// ---- POUs/Prototypes/TcoSequencer/TcoSequencerBase.TcPOU
(*~
        <docu>
            <summary>
                Provides basic sequential control, including step mode, which allows to run the sequence step-by-step, steping forward and steping backward.
            </summary>
        </docu>
~*)
FUNCTION_BLOCK ABSTRACT TcoSequencerBase EXTENDS TcoStateExtendible IMPLEMENTS ITcoSequencer, ITcoCoordinator
VAR CONSTANT
    MinStepID : INT := -32767;
    MaxStepID : INT := 32766;
    RESTORE_STEP_ID : INT := 32766;
END_VAR
VAR
    (*~
    <docu>
        <summary>
            Holds the status information about current step.
        </summary>
        <remarks>
            <para>
                See <see cref="StepDetails"/> for detailed description.
            </para>
        </remarks>
    </docu>
~*)
    {attribute addProperty Name "<#Current step#>"}
    _currentStep : StepDetails;
    (*~
    <docu>
        <summary>
            True if an error occurs in the sequence. Detailed cause of this error is described by the _sequencerErrorId.
        </summary>
        <remarks>
            <para>
                See <see cref="PlcDocu.TcoCore.TcoSequencer._sequencerErrorId"/> for detailed description.
            </para>
        </remarks>
    </docu>
~*)
    {attribute addProperty Name "<#Sequencer error#>"}
    {attribute clr [ReadOnly()]}
    _sequencerHasError : BOOL;
    (*~
    <docu>
        <summary>
            Describes cause of the sequencer error.
        </summary>
        <remarks>
            <para>
                See <see cref="TcoCore.eSequencerError"/> for detailed description.
            </para>
        </remarks>
    </docu>
~*)
    {attribute addProperty Name "<#Sequencer error ID#>"}
    {attribute clr [ReadOnly()]}
    _sequencerErrorId : eSequencerError := eSequencerError.noError;
    (*~
    <docu>
        <summary>
            Handles changing the sequencer mode (Cyclic, Step).
        </summary>
    </docu>
~*)
    _modeController : TcoSequencerModeController(THIS^);
    (*~
    <docu>
        <summary>
            Elapsed time of presently running sequence cycle.
        </summary>
    </docu>
~*)
    {attribute addProperty Name "<#Sequence cycle elapsed time#>"}
    _SequenceElapsedTime : TIME;
    (*~
    <docu>
        <summary>
            Elapsed time of the currently executing step.
        </summary>
    </docu>
~*)
    {attribute addProperty Name "<Current step time#>"}
    _StepElapsedTime : TIME;
    (*~
    <docu>
        <summary>
            Total time of the last sequence cycle.
        </summary>
    </docu>
~*)
    {attribute addProperty Name "<#Total sequence time#>"}
    _LastCycleTime : TIME;
END_VAR
VAR
    {attribute 'hide'}
    _isFirstStepEntry : BOOL;
    {attribute 'hide'}
    _theOrderOfTheCurrentlyEvaluatedStep : UINT;
    {attribute 'hide'}
    _theOrderOfTheCurrentlyExecutedStep : UINT;
    {attribute 'hide'}
    _theOrderOfThePreviouslyExecutedStep : UINT;
    {attribute 'hide'}
    _IdOfThePreviouslyExecutedStep : INT;
    {attribute 'hide'}
    _numberOfStepsInSequence : UINT;
    {attribute 'hide'}
    _previousNumberOfStepsInSequence : UINT;
    {attribute 'hide'}
    _stepCounter : UINT;
    {attribute 'hide'}
    _requestStepActive : BOOL;
    {attribute 'hide'}
    _requestedStepId : INT := MinStepID - 1;
    {attribute 'hide'}
    _cycleTimer : TON;
    {attribute 'hide'}
    _StepTimer : TON;
    {attribute 'hide'}
    _requestStepCycle : UINT;
    {attribute 'hide'}
    _StepIdChanged : BOOL;
    {attribute 'hide'}
    _StepOrderChanged : BOOL;
    {attribute 'hide'}
    _ChangeStepIdFrom : INT;
    {attribute 'hide'}
    _ChangeStepIdTo : INT;
    {attribute 'hide'}
    _ChangeStepOrderFrom : UINT;
    {attribute 'hide'}
    _ChangeStepOrderTo : UINT;
    {attribute 'hide'}
    _stepIdUniquenessChecked : BOOL := FALSE;
    {attribute 'hide'}
    _StepIdUniquenessControlState : eStepIdUniquenessControlState;
    {attribute 'hide'}
    _StepIdUniquenessStartCycleCount : ULINT;
    {attribute 'hide'}
    _checkStepIdRequestedInStepMode : BOOL;
    {attribute 'hide'}
    _restoringSequence : BOOL;
    {attribute 'hide'}
    _controlledStepIndex : UINT;
END_VAR
VAR
    {attribute 'hide'}
    _pPreviusSteps : POINTER TO INT;
END_VAR
VAR
    {attribute 'hide'}
    _lastOpeningCycle : ULINT;
    {attribute 'hide'}
    _lastClosingCycle : ULINT;
END_VAR
VAR
    _observer : ITcoSequencerObserver;
    {attribute 'hide'}
    _observerDummy : TcoTcoSequencerObserverDummy(THIS^);
END_VAR

METHOD PUBLIC FINAL ActivateDeveloperChecks
VAR_INPUT
END_VAR
IF (_StepIdUniquenessControlState = eStepIdUniquenessControlState.Deactivated) THEN
    _StepIdUniquenessControlState := eStepIdUniquenessControlState.Requested;
END_IF
END_METHOD

(*~
    <docu>
        <summary>
            Performs the check of the ```StepId``` of the currently executed step.
            <remarks>
                <note type="important">
                    The StepId of each step in the sequence must be unique throughout the complete sequence, and it must not be changed.
                    ```StepId``` sould be assigned as a number literal or a constant.
                </note>
            </remarks>
        </summary>
    </docu>
~*)
METHOD PRIVATE CheckStepId : BOOL
VAR_INPUT
    inStepID : INT;
    inStepModeActive : BOOL;
    inStepInRunning : BOOL;
END_VAR
CheckStepID := TRUE;

IF (_StepIdUniquenessControlState = eStepIdUniquenessControlState.Done) THEN
    IF ((_IdOfThePreviouslyExecutedStep <> inStepID) AND NOT _isFirstStepEntry AND (NOT inStepModeActive OR inStepInRunning)) THEN
        IF (_theOrderOfTheCurrentlyExecutedStep = 0) AND (_theOrderOfTheCurrentlyEvaluatedStep = 0) AND (_IdOfThePreviouslyExecutedStep = 0) THEN
            _IdOfThePreviouslyExecutedStep := inStepID;
        ELSIF NOT _StepIdChanged AND NOT _StepOrderChanged THEN
            _StepIdChanged := TRUE;
            _ChangeStepIdFrom := _IdOfThePreviouslyExecutedStep;
            _ChangeStepIdTo := inStepID;
            CheckStepID := FALSE;
        END_IF;
    END_IF
END_IF
END_METHOD

(*~
    <docu>
        <summary>
            Gets the information about the current step.
        </summary>
    </docu>
~*)
PROPERTY CurrentStep : REFERENCE TO StepDetails
GET
CurrentStep REF= _currentStep;
END_GET
END_PROPERTY

METHOD PUBLIC FINAL DeactivateDeveloperChecks
VAR_INPUT
END_VAR
_StepIdUniquenessControlState := eStepIdUniquenessControlState.Deactivated;
END_METHOD

{attribute 'hide'}
METHOD FB_init : BOOL
VAR_INPUT
    bInitRetains : BOOL; // if TRUE, the retain variables are initialized (warm start / cold start)
    bInCopyCode : BOOL; // if TRUE, the instance afterwards gets moved into the copy code (online change)
    ParentObject : ITcoObject;
    AutoRestoreMode : eRestoreMode;
END_VAR
END_METHOD

(*~
    <docu>
        <summary>
            Implicit call of this method is ensured by calling the method Run().
            It must not be called explicitely by consumer code in derived blocks.
            <remarks>
                <note type="important">
                    Do not call this method explicitly.
                </note>
            </remarks>
        </summary>
    </docu>
~*)
METHOD INTERNAL FINAL i_Close
_lastClosingCycle := Context.StartCycleCount;

IF _sequencerHasError THEN
    OnSequencerError(_sequencerErrorId);
END_IF

_previousNumberOfStepsInSequence := _numberOfStepsInSequence;
Context.Environment.Messaging.Suspend();

IF _modeController._stepIn.Done THEN
    _modeController._stepIn.Restore();
END_IF

Context.Environment.Messaging.Resume();
_restoringSequence := FALSE;
END_METHOD

(*~
    <docu>
        <summary>
            <para>
                Completes the sequencer, and return the sequencer pointer to the first step in the seuqence.
                Method is typically called inside the last step of the sequence.
            </para>
        </summary>
    </docu>
~*)
METHOD PROTECTED FINAL i_CompleteSequence
_theOrderOfTheCurrentlyExecutedStep := 0;
_LastCycleTime := _SequenceElapsedTime;
_cycleTimer(IN := FALSE, PT := T#0S);
_currentStep.Status := eStepStatus.Done;
OnSequenceCompleted();
OnStepCompleted();
Context.Environment.Messaging.Suspend();
_modeController._stepForward.Restore();
_modeController._stepBackward.Restore();
_modeController._stepIn.Restore();
Context.Environment.Messaging.Resume();
END_METHOD

(*~
    <docu>
        <summary>
            Completes the execution of the current step and moves the sequencer pointer to the next step in order of execution.
            The call returns `ITcoObjectRestorer` that allows to restore object upon step completition.
        </summary>
        <returns></returns>
    </docu>
~*)
METHOD PROTECTED FINAL i_CompleteStep : ITcoObjectRestorer
Messenger.Build()
    .Append('Leaving step id: ')
    .AppendAny(_currentStep.ID)
    .Append(' [')
    .Append(_currentStep.Description)
    .Append('] : ')
    .AppendAny(_theOrderOfTheCurrentlyExecutedStep)
    .As().AsTrace();

_theOrderOfTheCurrentlyExecutedStep := _theOrderOfTheCurrentlyExecutedStep + 1;
_currentStep.Status := eStepStatus.Done;
OnStepCompleted();
_modeController._stepIn.DoneWhen(_modeController._stepIn.Execute());
i_CompleteStep := THIS^;
END_METHOD

(*~
    <docu>
        <summary>
            Implicit calling of this method is ensured by calling the method Run().
            It must not be called explicitely by consumer code in derived blocks.
            <remarks>
                <note type="important">
                    Do not call this method explicitly.
                </note>
            </remarks>
        </summary>
    </docu>
~*)
METHOD INTERNAL FINAL i_Open
VAR
    _message : STRING(254);
END_VAR
_theOrderOfTheCurrentlyEvaluatedStep := 0;

IF _requestStepActive AND
    _requestedStepId <> (MinStepID - 1) AND
    (_modeController.Mode <> eSequencerMode.StepMode OR _modeController._stepIn.Busy OR _checkStepIdRequestedInStepMode) THEN
    _requestStepCycle := _requestStepCycle + 1;
ELSE
    _requestStepCycle := 0;
END_IF

IF _requestStepCycle > 1 AND NOT _sequencerHasError THEN
    _sequencerErrorId := eSequencerError.StepWithRequestedIdDoesNotExists;
    _message := CONCAT('REQUESTED STEP_ID: ', INT_TO_STRING(_requestedStepId));
    _message := CONCAT(_message, ' DOES NOT EXIST');
    _currentStep.Description := _message;
    _currentStep.Status := eStepStatus.Error;
    THIS^.Messenger.Post(_message, eMessageCategory.ProgrammingError);
    _sequencerHasError := TRUE;
END_IF

IF _StepIdUniquenessControlState = eStepIdUniquenessControlState.NotYetStarted OR
    _StepIdUniquenessControlState = eStepIdUniquenessControlState.Requested THEN
    _StepIdUniquenessControlState := eStepIdUniquenessControlState.Started;
END_IF;

_restoringSequence := FALSE;
_lastOpeningCycle := Context.StartCycleCount;
END_METHOD

(*~
    <docu>
        <summary>
            Terminates the currently executed step and set the sequencer's pointer to the step with Id that corresponds to ```inRequestedStepID``` parameter.
            When the order of the requested step is higher than the order of the currently finished step (the requested step is "after" the current one)
            the requested step is started in the same context cycle.
            When the order of the requested step is lower than the order of the currently finished step (the requested step is "before" the current one)
            the requested step is started in the next context cycle.
            If the requested step is not found even in the next context cycle, the sequencer enters error state ```StepWithRequestedIdDoesNotExists```.
            <para>
                See <see cref="TcoCore.eSequencerError"/> for detailed description.
            </para>
        </summary>
    </docu>
~*)
METHOD PROTECTED FINAL i_RequestStep : ITcoSequencer
VAR_INPUT
    (*~
        <docu>
            <summary>
                StepId of the step to be executed.
            </summary>
        </docu>
    ~*)
    inRequestedStepID : INT := MinStepID - 1;
END_VAR
VAR
    _message : STRING(254);
END_VAR
_modeController._stepIn.Restore();
_currentStep.Status := eStepStatus.Done;
_checkStepIdRequestedInStepMode := TRUE;

IF (inRequestedStepID <> (MinStepID - 1)) THEN
    IF _requestedStepId <> (MinStepID - 1) THEN
        IF NOT _sequencerHasError THEN
            _sequencerErrorId := eSequencerError.MultipleRequestStepMethodCall;
            _message := CONCAT('REQUESTED STEP_ID: ', INT_TO_STRING(inRequestedStepID));
            _message := CONCAT(_message, ' HAS BEEN REQUIRED, WHILE PREVIOUS REQUESTED STEP_ID: ');
            _message := CONCAT(_message, INT_TO_STRING(_requestedStepId));
            _message := CONCAT(_message, ' HAS NOT BEEN YET PERFORMED!');
            _currentStep.Description := _message;
            _currentStep.Status := eStepStatus.Error;
            THIS^.Messenger.Post(_message, eMessageCategory.ProgrammingError);
            _sequencerHasError := TRUE;
        END_IF
    ELSE
        _requestStepCycle := 0;
        _requestedStepId := inRequestedStepID;
        _requestStepActive := TRUE;
    END_IF
END_IF;

Messenger.Build()
    .Append('Leaving step id: ')
    .AppendAny(_currentStep.ID)
    .Append(' [')
    .Append(_currentStep.Description)
    .Append('] : ')
    .AppendAny(_theOrderOfTheCurrentlyExecutedStep)
    .As().AsTrace();

Messenger.Build().Append('Reqesting step id jump to: ').AppendAny(inRequestedStepID).As().AsTrace();
i_RequestStep := THIS^;
END_METHOD

(*~
    <docu>
        <summary>
                Step of the sequence.
                <note type="important">
                    Make sure you do not use the value of `32766` for the step id. This value is reserved for the restore step.
                <note>
        </summary>
        <returns>
            True when step with given `StepId` is in order of the execution; the step is enabled and the sequencer is in the cyclic mode.
            True when step with given `StepId` is in order of the execution; the step is enabled, the sequencer is in the step mode and StepIn() method has been triggered.
        </returns>
    </docu>
~*)
METHOD PROTECTED FINAL i_Step : BOOL
VAR_INPUT
    (*~
    <docu>
        <summary>
            StepId of the current step.
            <remarks>
                <note type="important">
                    This number must be unique throughout the complete sequence.
                    It must be a constant or numerical literal and it must not change during the life-time of the sequencer.
                </note>
                <note type="important">
                    Make sure you do not use the value of `32766` for the step id. This value is reserved for the restore step.
                <note>
            </remarks>
        </summary>
    </docu>
~*)
    inStepID : INT;
    (*~
    <docu>
        <summary>
            If this value is false, step body is not executed and execution is moved to the next enabled step.
        </summary>
    </docu>
~*)
    inEnabled : BOOL;
    (*~
    <docu>
        <summary>
            Step description text.
        </summary>
    </docu>
~*)
    inStepDescription : STRING(254);
END_VAR
VAR
    _message : STRING(254);
    _isInOrderOfExecution : BOOL;
    _stepModeActive : BOOL;
    _stepInExecuting : BOOL;
END_VAR
i_Step := FALSE;

IF inStepID < MinStepID THEN
    _message := CONCAT('STEP_ID TOO LOW: ', INT_TO_STRING(inStepID));
    _message := CONCAT(_message, '! MINIMAL VALUE POSSIBLE: ');
    _message := CONCAT(_message, INT_TO_STRING(MinStepID));
    _message := CONCAT(_message, '!!!');
    _currentStep.Description := _message;
    _currentStep.Status := eStepStatus.Error;
    THIS^.Messenger.Post(_message, eMessageCategory.ProgrammingError);
    _sequencerErrorId := eSequencerError.StepIdTooLow;
    _sequencerHasError := TRUE;
ELSIF inStepID > MaxStepID THEN
    _message := CONCAT('STEP_ID TOO HIGH: ', INT_TO_STRING(inStepID));
    _message := CONCAT(_message, '! MAXIMAL VALUE POSSIBLE: ');
    _message := CONCAT(_message, INT_TO_STRING(MaxStepID));
    _message := CONCAT(_message, '!!!');
    _currentStep.Description := _message;
    _currentStep.Status := eStepStatus.Error;
    THIS^.Messenger.Post(_message, eMessageCategory.ProgrammingError);
    _sequencerErrorId := eSequencerError.StepIdTooHigh;
    _sequencerHasError := TRUE;
ELSIF NOT _sequencerHasError THEN
    i_Step := StepInternal(inStepID, inEnabled, inStepDescription);
END_IF;

Observer.Observe(inIsStepActive := i_Step,
    inCurrentStepOrder := _theOrderOfTheCurrentlyExecutedStep,
    inID := inStepID,
    inOrder := _theOrderOfTheCurrentlyEvaluatedStep - 1,
    inEnabled := inEnabled,
    inDescription := inStepDescription,
    inStatus := _currentStep.Status,
    inDuration := _currentStep.Duration,
    inStepCount := _numberOfStepsInSequence);
END_METHOD

(*~
    <docu>
        <summary>
            Completes the actually running step, when the `inCondition` parameter is `TRUE`.
            Method is typically called inside a step as the transition method.
        </summary>
    </docu>
~*)
METHOD PROTECTED FINAL i_StepCompleteWhen
VAR_INPUT
    (*~
    <docu>
        <summary>
            The condition under which the step is completed.
        </summary>
    </docu>
~*)
    inCondition : BOOL;
END_VAR
IF (inCondition) THEN
    THIS^.i_CompleteStep();
END_IF
END_METHOD

(*~
    <docu>
        <summary>
            Gets `true` on the first entry into new state.
        </summary>
    </docu>
~*)
PROPERTY IsFreshState : BOOL
GET
IsFreshState := _isFirstStepEntry;
END_GET
END_PROPERTY

(*~
    <docu>
        <summary>
            Performs the check of the uniqueness of `inStepId` in the sequence.
            <remarks>
                <note type="important">
                    The StepId of each step in the sequence must be unique throughout the complete sequence, and it must not be changed.
                </note>
            </remarks>
        </summary>
    </docu>
~*)
METHOD PRIVATE IsStepIdUnique
VAR_INPUT
    (*~
    <docu>
        <summary>
            StepId to be checked for uniqueness.
        </summary>
    </docu>
~*)
    inStepID : INT;
END_VAR
VAR
    _i : UINT;
    _hiIndex : UINT;
    _pUid : INT;
    _pNewSteps : POINTER TO INT;
    _message : STRING(254);
END_VAR
//Change number of the steps in sequence detected
IF (_numberOfStepsInSequence <> _previousNumberOfStepsInSequence) AND
    _previousNumberOfStepsInSequence > 0 AND
    _stepIdUniquenessChecked AND
    (
    _StepIdUniquenessControlState = eStepIdUniquenessControlState.NotYetStarted OR _StepIdUniquenessControlState = eStepIdUniquenessControlState.Done
    ) THEN
    _StepIdUniquenessControlState := eStepIdUniquenessControlState.Requested;
END_IF

IF (_StepIdUniquenessControlState >= eStepIdUniquenessControlState.Started AND _StepIdUniquenessControlState < eStepIdUniquenessControlState.Done)
    THEN
    //If new PLC cycle was performed, step id uniqueness control is done
    IF _StepIdUniquenessControlState = eStepIdUniquenessControlState.Running AND
        THIS^.Context.StartCycleCount >= _StepIdUniquenessStartCycleCount + 1 THEN
        _stepIdUniquenessChecked := TRUE;
        _StepIdUniquenessControlState := eStepIdUniquenessControlState.Done;
        _numberOfStepsInSequence := _controlledStepIndex + 1;
    END_IF

    //If step id uniqueness control is finished, clear dynamic arrays
    IF _StepIdUniquenessControlState >= eStepIdUniquenessControlState.Done THEN
        IF (_pPreviusSteps <> 0) THEN
            __DELETE(_pPreviusSteps);
        END_IF

        IF (_pNewSteps <> 0) THEN
            __DELETE(_pNewSteps);
        END_IF

        RETURN;
    END_IF

    //First call with the very first step of the sequence
    IF _StepIdUniquenessControlState = eStepIdUniquenessControlState.Started THEN
        _StepIdUniquenessStartCycleCount := THIS^.Context.StartCycleCount;
        _controlledStepIndex := 0;

        //It should not exists, if yes delete and create again
        IF (_pPreviusSteps <> 0) THEN
            __DELETE(_pPreviusSteps);
        END_IF

        _pPreviusSteps := __NEW(UINT, 1);
        //Stores first StepId
        _pPreviusSteps[0] := inStepID;
        _StepIdUniquenessControlState := eStepIdUniquenessControlState.Running;
    ELSIF _StepIdUniquenessControlState = eStepIdUniquenessControlState.Running THEN
        // Increment order of the currently controlled step
        _controlledStepIndex := _controlledStepIndex + 1;

        IF (_pNewSteps <> 0) THEN
            __DELETE(_pNewSteps);
        END_IF

        _pNewSteps := __NEW(UINT, (_controlledStepIndex + 1));
        //Compare with previous Steps and copy previous Steps to new array
        _hiIndex := _controlledStepIndex - 1;

        FOR _i := 0 TO _hiIndex DO
            _pUid := _pPreviusSteps[_i];

            IF inStepID = _pUid THEN
                IF NOT _sequencerHasError THEN
                    _sequencerErrorId := eSequencerError.NotUniqueStepId;
                    _message := CONCAT('ERROR NOT UNIQUE STEP_ID ', INT_TO_STRING(inStepID));
                    _currentStep.Description := _message;
                    _currentStep.Status := eStepStatus.Error;
                    THIS^.Messenger.Post(_message, eMessageCategory.ProgrammingError);
                    _sequencerHasError := TRUE;
                    _StepIdUniquenessControlState := eStepIdUniquenessControlState.Error;
                    RETURN;
                END_IF
            ELSE
                _pNewSteps[_i] := _pPreviusSteps[_i];
            END_IF
        END_FOR
        //Store new StepId
        _pNewSteps[_controlledStepIndex] := inStepID;

        //Delete and create again
        IF (_pPreviusSteps <> 0) THEN
            __DELETE(_pPreviusSteps);
        END_IF

        _pPreviusSteps := __NEW(UINT, (_controlledStepIndex + 1));
        //Copy
        _hiIndex := _controlledStepIndex;

        FOR _i := 0 TO _hiIndex DO
            _pPreviusSteps[_i] := _pNewSteps[_i];
        END_FOR

        IF (_pNewSteps <> 0) THEN
            __DELETE(_pNewSteps);
        END_IF
    END_IF

    _numberOfStepsInSequence := _controlledStepIndex + 1;
END_IF
END_METHOD

(*~
    <docu>
        <summary>
            Main method of the sequener. Custom code needs to be placed here. The sequencer is executed by call of **Instance.Run()** method.
            This method is abstract, and it must be overridden in derived block.
        </summary>
    </docu>
~*)
METHOD PROTECTED ABSTRACT Main : BOOL
END_METHOD

(*~
    <docu>
        <summary>
            Handles changing the sequencer mode (Cyclic, Step).
        </summary>
    </docu>
~*)
PROPERTY ModeController : ITcoSequencerModeController
GET
ModeController := _modeController;
END_GET
END_PROPERTY

{attribute 'hide'}
{attribute 'obsolete' := 'You should access `MoveNext` via `ITcoCoordinator` interface.'}
METHOD PUBLIC MoveNext : BOOL
i_CompleteStep();
END_METHOD

(*~
    <docu>
        <summary>
            Get or sets the observer for this instance of the sequencer.
        </summary>
    </docu>
~*)
PROPERTY Observer : ITcoSequencerObserver
GET
IF (_observer <> 0) THEN
    Observer := _observer;
ELSE
    Observer := _observerDummy;
END_IF
END_GET
SET
_observer := Observer;
END_SET
END_PROPERTY

(*~
    <docu>
        <summary>
            Ensures that after each download, StepId uniqueness check is performed.
            <remarks>
                <note type="important">
                    Do not call this method explicitly.
                </note>
            </remarks>
        </summary>
    </docu>
~*)
{attribute 'call_after_online_change_slot' := '200'}
METHOD PRIVATE OnlineChange
IF _stepIdUniquenessChecked AND (_StepIdUniquenessControlState <> eStepIdUniquenessControlState.Deactivated) THEN
    _StepIdUniquenessControlState := eStepIdUniquenessControlState.Requested;
END_IF;
END_METHOD

(*~
    <docu>
        <summary>
            This method is called on sequence restore.
            This method can be overridden in derived block with a custom logic.
        </summary>
    </docu>
~*)
METHOD PROTECTED OnRestore
END_METHOD

(*~
    <docu>
        <summary>
            This method is called on sequence completion (the sequencer's last step was completed).
            This method can be overridden in derived block with a custom logic.
        </summary>
    </docu>
~*)
METHOD PROTECTED OnSequenceCompleted
END_METHOD

(*~
    <docu>
        <summary>
            This method is called when sequence enters error state. The method is called until the error is cleared.
            This method can be overridden in derived block with a custom logic.
        </summary>
    </docu>
~*)
METHOD PROTECTED OnSequencerError
VAR_INPUT
    inErrorId : eSequencerError;
END_VAR
END_METHOD

METHOD PROTECTED OnStateChange
VAR_INPUT
    PreviousState : INT;
    NewState : INT;
END_VAR
END_METHOD

(*~
    <docu>
        <summary>
            This method is executed upon step completion.
            This method can be overridden in derived block by custom logic.
        </summary>
    </docu>
~*)
METHOD PROTECTED OnStepCompleted
END_METHOD

(*~
    <docu>
        <summary>
            <para>
                This method resets the sequencer.
                Method is typically called before starting the sequence or after error has occured in the sequence.
            </para>
        </summary>
    </docu>
~*)
METHOD PUBLIC Restore : ITcoRestorable
_restoringSequence := TRUE;
_lastClosingCycle := 0;
_lastOpeningCycle := 0;
StepChanged(0);
_requestStepActive := FALSE;
_requestedStepId := MinStepID - 1;
_requestStepCycle := 0;
_sequencerHasError := FALSE;
_sequencerErrorId := eSequencerError.noError;
_currentStep.Description := '--------------------------';
_currentStep.ID := 0;
_currentStep.Order := 0;
_currentStep.Status := eStepStatus.None;
_currentStep.Duration := T#0S;
_stepCounter := 0;
_IdOfThePreviouslyExecutedStep := 0;
_numberOfStepsInSequence := 0;
_previousNumberOfStepsInSequence := 0;
_theOrderOfTheCurrentlyExecutedStep := 0;
_theOrderOfThePreviouslyExecutedStep := 0;
_stepIdUniquenessChecked := FALSE;
_StepIdUniquenessControlState := eStepIdUniquenessControlState.NotYetStarted;
_StepIdChanged := FALSE;
_StepOrderChanged := FALSE;
_ChangeStepIdFrom := 0;
_ChangeStepIdTo := 0;
_ChangeStepOrderFrom := 0;
_ChangeStepOrderTo := 0;
_StepTimer(IN := FALSE);
_cycleTimer(IN := FALSE);

IF _modeController.Mode = eSequencerMode.Invalid THEN
    _modeController.Mode := eSequencerMode.CyclicMode;
END_IF

Context.Environment.Messaging.Suspend();
_modeController._stepForward.Restore();
_modeController._stepBackward.Restore();
_modeController._stepIn.Restore();
Context.Environment.Messaging.Resume();
_checkStepIdRequestedInStepMode := FALSE;
OnRestore();
END_METHOD

{attribute 'hide'}
{attribute 'obsolete' := 'You should access `Retry` via `ITcoCoordinator` interface.'}
METHOD PUBLIC Retry : BOOL
VAR_INPUT
    inFromState : INT;
END_VAR
i_RequestStep(inFromState);
END_METHOD

(*~
    <docu>
        <summary>
            <para>
                Ensures calling the Open(), Main() and Close() methods in the desired order.
                This method is final, so it cannot be overloaded. The **Instance.Run()** needs to be called cyclically inside the appropriate context.
            </para>
        </summary>
    </docu>
~*)
METHOD PUBLIC ABSTRACT Run
END_METHOD

(*~
    <docu>
        <summary>
            This method is called at each transition between steps.
        </summary>
    </docu>
~*)
METHOD PRIVATE StepChanged
VAR_INPUT
    newState : INT;
END_VAR
_isFirstStepEntry := TRUE;
_theOrderOfThePreviouslyExecutedStep := 0;
_IdOfThePreviouslyExecutedStep := MinStepID - 1;
_StepTimer(IN := FALSE);
SUPER^.ChangeStateProtected(newState);
END_METHOD

(*~
    <docu>
        <summary>
                Basic step of the sequence.
        </summary>
        <returns>
            True in case when step with given StepId is in order of the execution, the step is enabled and the sequencer is in the cyclic mode.
            True in case when step with given StepId is in order of the execution, the step is enabled, the sequencer is in the step mode and StepIn() method was triggered.
        </returns>
    </docu>
~*)
METHOD PRIVATE StepInternal : BOOL
VAR_INPUT
    (*~
    <docu>
        <summary>
            StepId of the current step.
            <remarks>
                <note type="important">
                    This number must be unique throughout the complete sequence.
                    It must be a constant or numerical literal and it must not change during the life-time of the sequencer.
                </note>
            </remarks>
        </summary>
    </docu>
~*)
    inStepID : INT;
    (*~
    <docu>
        <summary>
            If this value is false, step body is not executed and execution is moved to the next enabled step.
        </summary>
    </docu>
~*)
    inEnabled : BOOL;
    (*~
    <docu>
        <summary>
            Step description text.
        </summary>
    </docu>
~*)
    inStepDescription : STRING(254);
END_VAR
VAR
    _message : STRING(254);
    _isInOrderOfExecution : BOOL;
    _stepModeActive : BOOL;
    _stepInExecuting : BOOL;
END_VAR
{warning disable C0195}
{warning disable C0196}
IF _modeController.Mode = eSequencerMode.Invalid THEN
    IF NOT _sequencerHasError THEN
        _currentStep.Description := 'INVALID MODE OF THE SEQUENCER!!!';
        _currentStep.Status := eStepStatus.Error;
        THIS^.Messenger.Post('INVALID MODE OF THE SEQUENCER!!!', eMessageCategory.Error);
        _sequencerErrorId := eSequencerError.InvalidSequencerMode;
        _sequencerHasError := TRUE;
    END_IF;

    RETURN;
END_IF
//-----------------------------------------------
//     		MULTIPLE CALL REGION
//-----------------------------------------------
// Initialize
StepInternal := FALSE;
_isFirstStepEntry := FALSE;

//-------------------------------------------------------------------------------------------------
//     		Check uniqueness of the StepId
//			If there are even two same StepIds or sequence has not been yet
//			checked, method return FALSE, so no entrance to the step will be executed
//-------------------------------------------------------------------------------------------------
//-------------------------------------------------------------------------------------------------
//In case of call Restore() in OnStateChange(), this method must exits
//otherwise we get page fault
IF _restoringSequence THEN
    RETURN;
END_IF

IsStepIDUnique(inStepID);

IF NOT _stepIdUniquenessChecked AND (_StepIdUniquenessControlState <> eStepIdUniquenessControlState.Deactivated) THEN
    //Produce StepChanged after first run of the first step
    {warning disable C0195}
    _theOrderOfThePreviouslyExecutedStep := -1;
    {warning enable C0195}
    RETURN;
END_IF
//-------------------------------------------------------------------------------------------------
//-------------------------------------------------------------------------------------------------
// Cycle time measurement
_cycleTimer(IN := TRUE, PT := T#48D40H62M47S295MS);
_SequenceElapsedTime := _cycleTimer.ET;

// Specific step request
IF (_requestStepActive) AND (_requestedStepId = inStepID) AND (_theOrderOfTheCurrentlyEvaluatedStep >= 0) THEN
    _currentStep.Status := eStepStatus.Done;
    _theOrderOfTheCurrentlyExecutedStep := _theOrderOfTheCurrentlyEvaluatedStep;
    _theOrderOfThePreviouslyExecutedStep := _theOrderOfTheCurrentlyExecutedStep;
    _requestedStepId := MinStepID - 1;
    _requestStepCycle := 0;
    _requestStepActive := FALSE;
    StepChanged(_requestedStepId);

    IF (inEnabled) THEN
        Messenger.Build()
            .Append('Entering step id: ')
            .AppendAny(inStepID)
            .Append(' [')
            .Append(inStepDescription)
            .Append('] : ')
            .AppendAny(_theOrderOfTheCurrentlyExecutedStep)
            .As().AsTrace();
    END_IF

    //In case of call Restore() in OnStateChange(), this method must exits
    //otherwise we get page fault
    IF NOT _stepIdUniquenessChecked THEN
        StepInternal := FALSE;
        RETURN;
    END_IF
END_IF

IF (_requestStepActive) THEN
    _theOrderOfTheCurrentlyEvaluatedStep := _theOrderOfTheCurrentlyEvaluatedStep + 1;
    RETURN;
END_IF
// STEP MODE COORDINATION
_stepModeActive := _modeController.Mode = eSequencerMode.StepMode;
_modeController(inCurrentStepRunning := _currentStep.Status = eStepStatus.Running);

IF (_stepModeActive) THEN
    // StepForward
    IF _modeController._stepForward.Execute() THEN
        _modeController._stepIn.Restore();
        _modeController._stepBackward.Restore();

        IF _theOrderOfTheCurrentlyExecutedStep < _numberOfStepsInSequence - 1 THEN
            _theOrderOfTheCurrentlyExecutedStep := _theOrderOfTheCurrentlyExecutedStep + 1;
            _modeController._stepForward.DoneWhen(TRUE);
        ELSE
            _modeController._stepForward.Restore();
        END_IF
    END_IF

    // Step Backward
    IF _modeController._stepBackward.Execute() THEN
        _modeController._stepIn.Restore();
        _modeController._stepForward.Restore();

        IF _theOrderOfTheCurrentlyExecutedStep > 0 THEN
            _theOrderOfTheCurrentlyExecutedStep := _theOrderOfTheCurrentlyExecutedStep - 1;
            _modeController._stepBackward.DoneWhen(TRUE);
        ELSE
            _modeController._stepForward.Restore();
        END_IF
    END_IF
END_IF;

Context.Environment.Messaging.Suspend();

IF (_modeController._stepForward.Done) THEN
    _modeController._stepForward.Restore();
END_IF

IF (_modeController._stepBackward.Done) THEN
    _modeController._stepBackward.Restore();
END_IF

Context.Environment.Messaging.Resume();
// Determine the step is in order of execution
_isInOrderOfExecution := (_theOrderOfTheCurrentlyExecutedStep = _theOrderOfTheCurrentlyEvaluatedStep);

//-----------------------------------------------
//     		SINGLE PER STEP CALL REGION
//-----------------------------------------------
IF (_StepIdUniquenessControlState = eStepIdUniquenessControlState.Deactivated) THEN
    _StepOrderChanged := FALSE;
    _StepIdChanged := FALSE;
    _sequencerHasError := FALSE;
END_IF

//Check if the order of the last executed step, has been changed
IF _StepIdUniquenessControlState = eStepIdUniquenessControlState.Done THEN
    IF (NOT _isInOrderOfExecution AND inStepID = _IdOfThePreviouslyExecutedStep) THEN
        IF _theOrderOfThePreviouslyExecutedStep <> _theOrderOfTheCurrentlyEvaluatedStep AND NOT _StepOrderChanged THEN
            _StepOrderChanged := TRUE;
            _ChangeStepOrderFrom := _theOrderOfThePreviouslyExecutedStep;
            _ChangeStepOrderTo := _theOrderOfTheCurrentlyEvaluatedStep;
        END_IF
    END_IF

    //Distinguish if StepId or step order has been changed
    IF (_theOrderOfTheCurrentlyEvaluatedStep >= (_stepCounter - 1)) AND _StepIdChanged OR _StepOrderChanged THEN
        IF _StepOrderChanged AND NOT _StepIdChanged THEN
            _message := CONCAT('ERROR, STEP ORDER CHANGED DURING STEP EXECUTION FROM: ', UINT_TO_STRING(_ChangeStepOrderFrom));
            _message := CONCAT(_message, '=>');
            _message := CONCAT(_message, UINT_TO_STRING(_ChangeStepOrderTo));
            _currentStep.Description := _message;
            _currentStep.Status := eStepStatus.Error;
            THIS^.Messenger.Post(_currentStep.Description, eMessageCategory.ProgrammingError);
            _sequencerErrorId := eSequencerError.OrderOfTheStepHasBeenChanged;
        ELSIF _StepOrderChanged AND _StepIdChanged AND (_ChangeStepOrderFrom = _ChangeStepIdTo) AND (_ChangeStepOrderTo = _ChangeStepIdFrom) THEN
            _message := CONCAT('ERROR, STEP ORDER CHANGED DURING STEP EXECUTION FROM: ', UINT_TO_STRING(_ChangeStepOrderFrom));
            _message := CONCAT(_message, '=>');
            _message := CONCAT(_message, UINT_TO_STRING(_ChangeStepOrderTo));
            _currentStep.Description := _message;
            _currentStep.Status := eStepStatus.Error;
            THIS^.Messenger.Post(_currentStep.Description, eMessageCategory.ProgrammingError);
            _sequencerErrorId := eSequencerError.OrderOfTheStepHasBeenChanged;
        ELSIF NOT _StepOrderChanged AND _StepIdChanged THEN
            _message := CONCAT('ERROR STEP_ID CHANGED DURING STEP EXECUTION FROM: ', UINT_TO_STRING(_ChangeStepIdFrom));
            _message := CONCAT(_message, '=>');
            _message := CONCAT(_message, UINT_TO_STRING(_ChangeStepIdTo));
            _currentStep.Description := _message;
            _currentStep.Status := eStepStatus.Error;
            THIS^.Messenger.Post(_currentStep.Description, eMessageCategory.ProgrammingError);
            _sequencerErrorId := eSequencerError.StepIdHasBeenChanged;
        ELSIF _StepOrderChanged AND _StepIdChanged AND (_ChangeStepOrderFrom = _ChangeStepIdFrom) AND (_ChangeStepOrderTo = _ChangeStepIdTo) THEN
            _message := CONCAT('ERROR STEP_ID CHANGED DURING STEP EXECUTION FROM: ', UINT_TO_STRING(_ChangeStepIdFrom));
            _message := CONCAT(_message, '=>');
            _message := CONCAT(_message, UINT_TO_STRING(_ChangeStepIdTo));
            _currentStep.Description := _message;
            _currentStep.Status := eStepStatus.Error;
            THIS^.Messenger.Post(_currentStep.Description, eMessageCategory.ProgrammingError);
            _sequencerErrorId := eSequencerError.StepIdHasBeenChanged;
        END_IF

        _sequencerHasError := TRUE;
    END_IF

    IF NOT _isInOrderOfExecution AND _StepIdChanged THEN
        _theOrderOfTheCurrentlyEvaluatedStep := _theOrderOfTheCurrentlyEvaluatedStep + 1;
    END_IF

    IF (_StepOrderChanged OR _StepIdChanged OR _sequencerHasError) THEN
        RETURN;
    END_IF
END_IF

IF (_isInOrderOfExecution AND NOT (_currentStep.Status = eStepStatus.Error)) THEN
    _currentStep.Status := eStepStatus.ReadyToRun;

    // Step is in the order of the execution, but it is disabled
    IF NOT inEnabled THEN
        _currentStep.Status := eStepStatus.Disabled;
    END_IF

    _stepInExecuting := _modeController._stepIn.Busy;

    IF (NOT inEnabled AND NOT _stepInExecuting AND NOT _stepModeActive) THEN
        _theOrderOfTheCurrentlyExecutedStep := _theOrderOfTheCurrentlyExecutedStep + 1;
    END_IF

    IF _stepModeActive THEN
        IF _modeController._stepIn.Execute() THEN
            _stepInExecuting := TRUE;

            // Skips the step when not enabled
            IF (NOT inEnabled) THEN
                _theOrderOfTheCurrentlyExecutedStep := _theOrderOfTheCurrentlyExecutedStep + 1;
                _modeController._stepIn.Restore();
            END_IF
        END_IF

        _currentStep.ID := inStepID;
        _currentStep.Enabled := inEnabled;

        IF NOT inEnabled THEN
            _currentStep.Description := CONCAT('(*', inStepDescription);
            _currentStep.Description := CONCAT(_currentStep.Description, '*)');
        ELSE
            _currentStep.Description := CONCAT('(>', inStepDescription);
            _currentStep.Description := CONCAT(_currentStep.Description, '<)');
        END_IF
    END_IF

    StepInternal := (NOT _stepModeActive OR _stepInExecuting) AND inEnabled AND NOT (_currentStep.Status = eStepStatus.Error);

    Messenger.OnCondition((NOT _stepModeActive OR _stepInExecuting) AND NOT inEnabled)
        .Build()
        .Append('Skipping disabled step id: ')
        .AppendAny(inStepID)
        .Append(' [')
        .Append(inStepDescription)
        .Append('] : ')
        .AppendAny(_theOrderOfTheCurrentlyExecutedStep)
        .As().AsTrace();

    IF (StepInternal) THEN
        //First entry to step production
        IF (_theOrderOfThePreviouslyExecutedStep <> _theOrderOfTheCurrentlyExecutedStep) THEN
            _isFirstStepEntry := TRUE;
            StepChanged(inStepID);

            //In case of call Restore() in OnStateChange(), this method must exits
            //otherwise we get page fault
            IF NOT _stepIdUniquenessChecked AND (_StepIdUniquenessControlState <> eStepIdUniquenessControlState.Deactivated) THEN
                StepInternal := FALSE;
                RETURN;
            END_IF
        END_IF;

        IF NOT CheckStepID(inStepID, _stepModeActive, _stepInExecuting) THEN
            StepInternal := FALSE;
            _theOrderOfTheCurrentlyEvaluatedStep := _theOrderOfTheCurrentlyEvaluatedStep + 1;
            _currentStep.Status := eStepStatus.Error;
            RETURN;
        END_IF

        _StepTimer(IN := StepInternal, PT := T#48D);
        _StepElapsedTime := _StepTimer.ET;
        _currentStep.ID := inStepID;
        _currentStep.Enabled := inEnabled;
        _currentStep.Description := inStepDescription;
        _currentStep.Duration := _StepElapsedTime;
        _IdOfThePreviouslyExecutedStep := inStepID;
        _theOrderOfThePreviouslyExecutedStep := _theOrderOfTheCurrentlyExecutedStep;
        _currentStep.Status := eStepStatus.Running;
        _currentStep.Order := _theOrderOfTheCurrentlyExecutedStep;

        Messenger.Build()
            .Append('Entering step id: ')
            .AppendAny(inStepID)
            .Append(' [')
            .Append(inStepDescription)
            .Append('] : ')
            .AppendAny(_theOrderOfTheCurrentlyExecutedStep)
            .As().AsTrace();
    END_IF
END_IF
//-----------------------------------------------
//     		CONTINUOUS CALL REGION
//-----------------------------------------------
// Increment flow number
_theOrderOfTheCurrentlyEvaluatedStep := _theOrderOfTheCurrentlyEvaluatedStep + 1;

IF (_stepCounter < _theOrderOfTheCurrentlyEvaluatedStep) THEN
    _stepCounter := _theOrderOfTheCurrentlyEvaluatedStep;
END_IF

_numberOfStepsInSequence := _stepCounter;
{warning enable C0195}
{warning enable C0196}
END_METHOD

{attribute 'hide'}
{attribute 'obsolete' := 'You should access `Terminate` via `ITcoCoordinator` interface.'}
METHOD PUBLIC Terminate : BOOL
VAR_INPUT
END_VAR
i_RequestStep(RESTORE_STEP_ID);
END_METHOD

END_FUNCTION_BLOCK

// ---- POUs/Prototypes/TcoState/TcoStateExtendible.TcPOU
FUNCTION_BLOCK ABSTRACT TcoStateExtendible EXTENDS TcoStateBase

METHOD PROTECTED FINAL ChangeState : ITcoState
VAR_INPUT
    NewState : INT;
END_VAR
ChangeState := SUPER^.ChangeStateProtected(NewState);
END_METHOD

(*~
    <docu>
        <summary>
            This method is called on each change of the <c>State</c>. This method could be overloaded and custom code should be placed here.
        </summary>
    </docu>
~*)
METHOD PROTECTED OnStateChange
VAR_INPUT
    PreviousState : INT;
    NewState : INT;
END_VAR
SUPER^.OnStateChange(PreviousState, NewState);
END_METHOD

END_FUNCTION_BLOCK

// ---- POUs/Prototypes/TcoState/TcoStateBase.TcPOU
(*~
    <docu>
        <summary>
            Provides basic state controller. It could be implemented using <c>IF</c>, <c>IF</c> <c>ELSIF</c> or <c>CASE</c> statement. The transition to the different state needs to be perfromed by calling
            <see cref="PlcDocu.TcoCore.TcoStateBase.ChangeState(Object)"/> method. This method ensures also calling the <see cref="PlcDocu.TcoCore.TcoStateBase.OnStateChange(Object,Object)"/> every time that state is changed. The
              <c>OnStateChange()</c>could be overloaded and some custom code that needs to be executed on each change of the state could be placed here. The TcoState could be used like this:
            <para>
                <example>
                <note type="Example 1">
                <para>
                    <c>_myTask()</c> is not a member of this <c>TcoState()</c>, it is restored manually to be able to trigger it in the next state.
                </para>
                    <code>
                        IF State = 10 THEN
                            Main._myTask.Invoke();
                            Main._myTask.Execute();
                            IF Main._myTask.Done THEN
                                ChangeState(State + 10);
                                Main._myTask.Restore();
                            END_IF
                        END_IF
                        IF State = 20 THEN
                            Main._myTask.Invoke();
                            Main._myTask.Execute();
                            IF Main._myTask.Done THEN
                                ChangeState(State + 10);
                                Main._myTask.Restore();
                            END_IF
                        END_IF
                    </code>
                 </note>
                </example>
            </para>
            <para>
                <example>
                <note type="Example 2">
                <para>
                    <c>_myTask()</c> is a member of this <c>TcoState()</c>, it is restored manually using the fluent syntax to be able to trigger it in the next state.
                </para>
                    <code>
                        CASE State OF
                            10:
                            _myTask.Invoke();
                            _myTask.Execute();
                            IF _myTask.Done THEN
                                ChangeState(State + 10).RestoreObject(_myTask);
                            END_IF
                            20:
                            _myTask.Invoke();
                            _myTask.Execute();
                            IF _myTask.Done THEN
                                ChangeState(State + 10).RestoreObject(_myTask);
                            END_IF
                        END_CASE
                    </code>
                 </note>
                </example>
                <para>
                    See <see cref="PlcDocu.TcoCore.TcoState.RestoreObject(Object)"/> for more details.
                </para>
            </para>
        </summary>
    </docu>
~*)
FUNCTION_BLOCK ABSTRACT TcoStateBase EXTENDS TcoObject IMPLEMENTS ITcoState, ITcoObjectRestorer
VAR
    {attribute clr [ReadOnly()]}
    _State : INT;
    {attribute 'hide'}
    _enableAutoRestore : BOOL;
    {attribute 'hide'}
    _AutoRestorable : BOOL;
    {attribute 'hide'}
    _StartCycleCount : ULINT;
    {attribute 'hide'}
    _MyParentsChangeStateCycle : ULINT;
    {attribute 'hide'}
    _ChangeStateCycle : ULINT;
    {attribute 'hide'}
    _LastChangedState : INT;
    {attribute 'hide'}
    _MyParentsLastChangedState : INT;
END_VAR

(*~
    <docu>
        <summary>
            Returns if this instance is auto restorable. This is 'dependency property'. Value of this property is given by the parent of this object.
            This value is assigned after download by calling the implicit method <c>FB_init()</c> of the parent object and cannot be changed during runtime.
            The <c>AutoRestorable</c> property of this objects is retrieved from the <c>EnableAutoRestore</c> property of the parent object.
            This is done by calling the <c>CheckIfAutoRestoreEnabledByParent()</c> method inside the implicit method <c>FB_init()</c> after download.
            If this instance is the auto restorable it will call the <see cref="PlcDocu.TcoCore.TcoState.Restore()"/> method if:
            <para>
                1.) This instance has not been called for one or more cycles and starts to be called again. (By calling the instance means asking for its property <see cref="PlcDocu.TcoCore.TcoState.State()"/> property).
            </para>
            <para>
                2.)	Parent object of this instance changes its state.
            </para>
            <para>
                See also <see cref="PlcDocu.TcoCore.TcoState.EnableAutoRestore()"/>
            </para>
        </summary>
    </docu>
~*)
PROPERTY AutoRestorable : BOOL
GET
AutoRestorable := _AutoRestorable;
END_GET
END_PROPERTY

(*~
    <docu>
        <summary>
            Private method called each time that State property is asked for. If this instance is auto restorable, this method ensures calling the <see cref="PlcDocu.TcoCore.TcoState.Restore()"/> method if:
            <para>
                1.)	Parent object of this instance changes its state in this Plc cycle.
            </para>
            <para>
                2.)	Parent object of this instance changes its state no mather when and this instance has not yet process this change.
            </para>
            <para>
                3.) This instance has not been called for one or more cycles and starts to be called again. (By calling the instance means asking for its property <see cref="PlcDocu.TcoCore.TcoState.State()"/> property).
            </para>
            <para>
                See also <see cref="PlcDocu.TcoCore.TcoState.AutoRestorable()"/>
            </para>
            <para>
                See also <see cref="PlcDocu.TcoCore.TcoState.EnableAutoRestore()"/>
            </para>
        </summary>
    </docu>
~*)
METHOD PRIVATE AutoRestore
VAR
    _MyParent_TcoState : ITcoState := 0;
    _MyParent_ChangeStateCycle : ULINT;
    _MyParent_LastChangeState : INT;
END_VAR
//If parent of this instance is TcoState type or its derived type and the parent
//EnableAutoRestore property is set to TRUE, this instance determines the value
//of its own AutoRestorable property by calling CheckIfAutoRestoreEnabledByParent
//after each download.
IF _AutoRestorable THEN
    IF __QUERYINTERFACE(THIS^.Parent, _MyParent_TcoState) THEN
        _MyParent_ChangeStateCycle := _MyParent_TcoState.LastStateChangeCycle;
        _MyParent_LastChangeState := _MyParent_TcoState.State;
    END_IF;

    //If OnStateChange event of the parent has occured, the value of the parent's
    //StartCycleCount property is stored into its ChangeStateCycle property.
    //Each child has to deal with it individually in the next call of its body,
    //restore itself, and copy the parent's ChangeStateCycle property into the
    //child's own property.
    IF _MyParent_ChangeStateCycle <> _MyParentsChangeStateCycle THEN
        THIS^.Restore();
        _MyParentsChangeStateCycle := _MyParent_ChangeStateCycle;
    END_IF

    IF _MyParent_LastChangeState <> _MyParentsLastChangedState THEN
        THIS^.Restore();
        _MyParentsLastChangedState := _MyParent_LastChangeState;
    END_IF
END_IF
END_METHOD

(*~
    <docu>
        <summary>
            Use to change the State property of this instance to the new value. This method is final, so it cannot be overloaded. However there is a <see cref="PlcDocu.TcoCore.TcoState.OnStateChange(Object,Object)"/>
            method that is called on each change of the <c>State</c> and could be overloaded.
            <para>
                <example>
                <note type="Example">
                <para>
                    Possibility to use the fluent syntax.
                </para>
                    <code>ChangeState(newState).RestoreObject(myChildObject);</code>
                 </note>
                </example>
            </para>
        </summary>
    </docu>
~*)
METHOD PROTECTED ChangeStateProtected : ITcoState
VAR_INPUT
    NewState : INT;
END_VAR
VAR
    PreviousState : INT;
END_VAR
PreviousState := THIS^._State;
THIS^._State := NewState;

IF NewState <> PreviousState THEN
    _ChangeStateCycle := THIS^.Context.StartCycleCount;
    _LastChangedState := NewState;
    THIS^.OnStateChange(PreviousState, NewState);
END_IF;

ChangeStateProtected := THIS^;
END_METHOD

(*~
    <docu>
        <summary>
            This method ensures reading out the parent's <see cref="PlcDocu.TcoCore.TcoStateBase.EnableAutoRestore()/> property and writing it into the <see cref="PlcDocu.TcoCore.TcoStateBase.AutoRestorable()"/> of this instance.
            Calling this method is ensured by calling the implicit method <c>FB_init()</c> after download, or after online change.
        </summary>
    </docu>
~*)
{attribute 'call_after_online_change_slot' := '100'}
METHOD PRIVATE CheckIfAutoRestoreEnabledByParent
VAR
    _MyParent_TcoState : ITcoState := 0;
END_VAR
IF __QUERYINTERFACE(THIS^.Parent, _MyParent_TcoState) THEN
    _AutoRestorable := _MyParent_TcoState.IsAutoRestoreEnabled;
END_IF;
END_METHOD

(*~
    <docu>
        <summary>
            Private method called each time that the <see cref="PlcDocu.TcoCore.TcoStateBase.State()"/> property is asked for.
            If this instance is auto restorable, this method ensures calling the <see cref="PlcDocu.TcoCore.TcoStateBase.Restore()"/> method if
            this instance has not been called for one or more cycles and starts to be called again. (By calling the instance means asking for its property State).
            <para>
                See also <see cref="PlcDocu.TcoCore.TcoStateBase.AutoRestorable"/>
            </para>
            <para>
                See also <see cref="PlcDocu.TcoCore.TcoStateBase.EnableAutoRestore"/>
            </para>
        </summary>
    </docu>
~*)
METHOD PRIVATE CheckIfCalledCyclically
VAR
    _MyContextStartCycleCount : ULINT;
END_VAR
//If parent of this instance is TcoState type or its derived type and the parent
//EnableAutoRestore property is set to TRUE, this instance determines the value
//of its own AutoRestorable property by calling CheckIfAutoRestoreEnabledByParent
//after each download.
IF _AutoRestorable THEN
    _MyContextStartCycleCount := THIS^.Context.StartCycleCount;

    //If this instance is AutoRestorable, its body has to be called cyclically,
    //otherwise this instance is restored.
    //This mechanism force the user to call this instance properly,
    //in order to don't miss the OnStateChange() event of the parent
    //in case of the body of this instance isn't called.
    IF _MyContextStartCycleCount > _StartCycleCount + 1 THEN
        THIS^.Restore();
    END_IF

    _StartCycleCount := _MyContextStartCycleCount;
END_IF
END_METHOD

(*~
    <docu>
        <summary>
            Returns the context of the parent object, that this object is assigned to.
            This context is given by declaration, its value is assigned after download by calling the implicit method <c>FB_init()</c> and cannot be changed during runtime.
        </summary>
    </docu>
~*)
PROPERTY Context : ITcoContext
GET
Context := THIS^.Parent.Context;
END_GET
END_PROPERTY

{attribute 'hide'}
METHOD FB_init : BOOL
VAR_INPUT
    bInitRetains : BOOL; // if TRUE, the retain variables are initialized (warm start / cold start)
    bInCopyCode : BOOL; // if TRUE, the instance afterwards gets moved into the copy code (online change)
    ParentObject : ITcoObject;
    AutoRestoreMode : eRestoreMode;
END_VAR
_Identity := ADR(THIS^);
_ParentObject := ParentObject;
_enableAutoRestore := AutoRestoreMode = eRestoreMode.AutoRestoreMembers;
CheckIfAutoRestoreEnabledByParent();
END_METHOD

(*~
    <docu>
        <summary>
            Returns the identity of the this object.
            This variable is used in the higher level packages.
        </summary>
    </docu>
~*)
PROPERTY Identity : ULINT
GET
Identity := _Identity;
END_GET
END_PROPERTY

(*~
    <docu>
        <summary>
            Returns if the auto restore mechanism is enabled for this instance. This property does not affect this instance, but it affects all members of this instance.
            If the auto restore is enabled, the child member call its <c>Restore()</c> method if:
            <para>
            1.) Its instance has not been called for one or more cycles.
            </para>
            <para>
            2.)	Its parent object (THIS^ instance) has changed its state.
            </para>
            This value is assigned after download by calling the implicit method <c>FB_init()</c> and cannot be changed during runtime.
            <para>
                See also <see cref="PlcDocu.TcoCore.TcoStateBase.AutoRestorable()"/>
            </para>
        </summary>
    </docu>
~*)
PROPERTY IsAutoRestoreEnabled : BOOL
GET
IsAutoRestoreEnabled := _enableAutoRestore;
END_GET
END_PROPERTY

(*~
    <docu>
        <summary>
            Returns number of the Plc cycle during which this instance changes its <c>State</c> last time.
            The child objects ask for this value to ensure auto restore mechanism working.
        </summary>
    </docu>
~*)
PROPERTY LastStateChangeCycle : ULINT
GET
LastStateChangeCycle := _ChangeStateCycle;
END_GET
END_PROPERTY

(*~
    <docu>
        <summary>
            This method is called on each change of the <c>State</c>. This method could be overloaded and custom code should be placed here.
        </summary>
    </docu>
~*)
METHOD PROTECTED OnStateChange
VAR_INPUT
    PreviousState : INT;
    NewState : INT;
END_VAR
END_METHOD

(*~
    <docu>
        <summary>
            Restores this instance to the state -1.
            <para>
                <example>
                    <note type="Example">
                        <para>
                            Possibility to use the fluent syntax.
                        </para>
                        <code>
                            Restore().RestoreObject(myFirstChildObject).RestoreObject(mySecondChildObject);
                        </code>
                     </note>
                </example>
            </para>
            <para>
                See also <see cref="PlcDocu.TcoCore.TcoState.AutoRestorable()"/>
            </para>
            <para>
                See also <see cref="PlcDocu.TcoCore.TcoState.EnableAutoRestore()"/>
            </para>
        </summary>
    </docu>
~*)
METHOD Restore : ITcoRestorable
ChangeStateProtected(-1);
Restore := THIS^;
END_METHOD

(*~
    <docu>
        <summary>
            Ensures the call of the <c>Restore()</c> method in fluent-like fashion.
            <para>
                <example>
                <note type="Example">
                <para>
                    Possibility to use the fluent syntax.
                </para>
                    <code>ChangeState(newState).RestoreObject(myFirstChildObject).RestoreObject(mySecondChildObject);</code>
                 </note>
                </example>
            </para>
        </summary>
    </docu>
~*)
METHOD RestoreObject : ITcoObjectRestorer
VAR_INPUT
    Obj : ITcoRestorable;
END_VAR
Obj.Restore();
RestoreObject := THIS^;
END_METHOD

(*~
    <docu>
        <summary>
            Return actual state of this instance. Needs to be asked for cyclically in case of this instance is auto restorable.
            <para>
                See also <see cref="PlcDocu.TcoCore.TcoStateBase.AutoRestorable()"/>
            </para>
        </summary>
    </docu>
~*)
PROPERTY State : INT
GET
CheckIfCalledCyclically();
AutoRestore();
State := _State;
END_GET
END_PROPERTY

END_FUNCTION_BLOCK

// ---- POUs/Prototypes/TcoSequencer/TcoSequencerModeController.TcPOU
(*~
        <docu>
            <summary>
                Provides switching between sequencer modes so as handling stepping tasks in the step mode.
            </summary>
        </docu>
~*)
FUNCTION_BLOCK TcoSequencerModeController EXTENDS TcoObject IMPLEMENTS ITcoSequencerModeController
VAR_INPUT
    inCurrentStepRunning : BOOL;
END_VAR
VAR
    (*~
    <docu>
        <summary>
            When `TRUE`, disables changing between the modes of the sequencer.
        </summary>
    </docu>
~*)
    {attribute addProperty Name "<#Changing mode disabled#>"}
    {attribute clr [ReadOnly()]}
    _DisableModeChanging : BOOL;
    (*~
    <docu>
        <summary>
            When `TRUE` skipping steps of the sequencer using methods `StepBackward()` and `StepForward()` is disabled.
        </summary>
    </docu>
~*)
    {attribute addProperty Name "<#Skipping steps disabled#>"}
    {attribute clr [ReadOnly()]}
    _DisableStepSkipping : BOOL;
    (*~
    <docu>
        <summary>
            Triggers StepBackward task, that decrements current step (variable: <c> TcoSequencer._theOrderOfTheCurrentlyExecutedStep</c> ), in case the sequencer is in step mode, and the current step is greather than zero.
        </summary>
    </docu>
~*)
    {attribute addProperty Name "<#Step backward#>"}
    _stepBackward : TcoTask(THIS^);
    (*~
    <docu>
        <summary>
            Triggers StepIn task, that changes the current step status from ReadyToRun to Running.
            This causes starting the execution of the body of the current step.
        </summary>
    </docu>
~*)
    {attribute addProperty Name "<#Step in#>"}
    _stepIn : TcoTask(THIS^);
    (*~
    <docu>
        <summary>
            Triggers StepForward task, that increment current step (variable: <c>TcoSequencer._theOrderOfTheCurrentlyExecutedStep</c> ),
            in case the sequencer is in step mode, and the current step is lower than number of steps in th sequence (variable: <c>TcoSequencer._numberOfStepsInSequence</c> ).
        </summary>
    </docu>
~*)
    {attribute addProperty Name "<#Step forward#>"}
    _stepForward : TcoTask(THIS^);
    (*~
    <docu>
        <summary>
            Toggles between cyclic mode and step mode if not disabled.
            <para>
                See <see cref="PlcDocu.TcoCore.TcoSequencerModeController.DisableModeChanging()"/> for detailed description.
            </para>
        </summary>
    </docu>
~*)
    {attribute addProperty Name "<#Change mode#>"}
    _changeMode : TcoTask(THIS^);
    (*~
    <docu>
        <summary>
            Current mode of the sequencer.
        </summary>
    </docu>
~*)
    {attribute addProperty Name "<#Mode#>"}
    {attribute clr [ReadOnly()]}
    _mode : eSequencerMode;
    {attribute 'hide'}
    _previousMode : eSequencerMode := eSequencerMode.Invalid;
END_VAR

THIS^._changeMode.Enabled := NOT _DisableModeChanging;

IF _changeMode.Execute() THEN
    IF Mode = eSequencerMode.CyclicMode THEN
        Mode := eSequencerMode.StepMode;
        _changeMode.Restore();
        RETURN;
    END_IF

    IF Mode = eSequencerMode.StepMode THEN
        Mode := eSequencerMode.CyclicMode;
        _changeMode.Restore();
        RETURN;
    END_IF
END_IF

ChangeMode();

IF _changeMode.Done OR _changeMode.Error THEN
    _changeMode.Restore();
END_IF

METHOD PRIVATE ChangeMode
IF _previousMode <> _mode THEN
    //Restore all stepping task on mode change
    _stepForward.Restore();
    _stepBackward.Restore();
    _stepIn.Restore();
    _changeMode.Restore();

    //Mode change from cyclic to step, enabling stepping tasks according to settings.
    IF _previousMode = eSequencerMode.CyclicMode AND _mode = eSequencerMode.StepMode THEN
        _stepBackward.Enabled := NOT THIS^._DisableStepSkipping;
        _stepIn.Enabled := TRUE;
        _stepForward.Enabled := NOT THIS^._DisableStepSkipping;

        //If current step was running at the moment of switching from cyclic to step, stepIn task is invoked.
        IF inCurrentStepRunning THEN
            _stepIn.Invoke();
        END_IF
    END_IF

    //Disabling stepping tasks in case of Cyclic mode.
    IF _mode = eSequencerMode.CyclicMode THEN
        _stepBackward.Enabled := FALSE;
        _stepIn.Enabled := FALSE;
        _stepForward.Enabled := FALSE;
    END_IF

    _previousMode := _mode;
    OnModeChange(_previousMode, _mode);
END_IF
END_METHOD

(*~
    <docu>
        <summary>
            When ```TRUE```, disables mode change.
        </summary>
    </docu>
~*)
PROPERTY DisableModeChanging : BOOL
GET
DisableModeChanging := _DisableModeChanging;
END_GET
SET
_DisableModeChanging := DisableModeChanging;
END_SET
END_PROPERTY

(*~
    <docu>
        <summary>
            When ```TRUE``` disables step skipping (```StepBackward()``` and ```StepForward()```).
        </summary>
    </docu>
~*)
PROPERTY DisableStepSkipping : BOOL
GET
DisableStepSkipping := _DisableStepSkipping;
END_GET
SET
_DisableStepSkipping := DisableStepSkipping;
END_SET
END_PROPERTY

(*~
    <docu>
        <summary>
            Gets or sets the mode of the sequencer.
        </summary>
    </docu>
~*)
PROPERTY Mode : eSequencerMode
GET
Mode := _mode;
END_GET
SET
IF NOT _DisableModeChanging THEN
    _mode := Mode;
END_IF
END_SET
END_PROPERTY

(*~
    <docu>
        <summary>
            Executes when mode of the sequencer changes.
        </summary>
    </docu>
~*)
METHOD PROTECTED OnModeChange
VAR_INPUT
    PreviousMode : eSequencerMode;
    NewMode : eSequencerMode;
END_VAR
END_METHOD

(*~
    <docu>
        <summary>
            Moves the sequencers pointer to the previous step.
        </summary>
    </docu>
~*)
METHOD PUBLIC FINAL StepBackward
_stepBackward.Invoke();
END_METHOD

(*~
    <docu>
        <summary>
            Moves the sequencers pointer to the next step.
        </summary>
    </docu>
~*)
METHOD PUBLIC FINAL StepForward
_stepForward.Invoke();
END_METHOD

(*~
    <docu>
        <summary>
            Executes the step at the current sequencer's pointer.
        </summary>
    </docu>
~*)
METHOD PUBLIC FINAL StepIn
_stepIn.Invoke();
END_METHOD

END_FUNCTION_BLOCK

// ---- POUs/Prototypes/TcoSequencer/TcoSequencerObserver/TcoTcoSequencerObserverDummy.TcPOU
FUNCTION_BLOCK INTERNAL TcoTcoSequencerObserverDummy EXTENDS TcoObject IMPLEMENTS ITcoSequencerObserver

METHOD Observe
VAR_INPUT
    (*~
    <docu>
        <summary>
            Indicates that a step is active.
        </summary>
    </docu>
    ~*)
    inIsStepActive : BOOL;
    (*~
    <docu>
        <summary>
            Currently running step order.
        </summary>
    </docu>
    ~*)
    inCurrentStepOrder : UINT;
    (*~
    <docu>
        <summary>
            Step identification number.
        </summary>
        <remarks>
             <note type="important">
                This number must be unique throughout the complete sequence. It is required to uniquely identify the step of the sequence.
            </note>
            <para>
                The <see cref="PlcDocu.TcoCore.TcoSequencer.RequestStep"/> method is using this number to jump to the required step.
            </para>
        </remarks>
    </docu>
    ~*)
    {attribute addProperty Name "<#Step ID#>"}
    inID : INT;
    (*~
        <docu>
            <summary>
                Order of the step in the sequence.
            </summary>
        </docu>
    ~*)
    {attribute addProperty Name "<#Step Order#>"}
    inOrder : UINT;
    (*~
        <docu>
            <summary>
                If this value is false, step body is not executed and execution is moved to the next enabled step in the sequence.
            </summary>
        </docu>
    ~*)
    {attribute addProperty Name "<#Enabled#>"}
    inEnabled : BOOL;
    (*~
        <docu>
            <summary>
                Step description text.
            </summary>
        </docu>
    ~*)
    {attribute addProperty Name "<#Step description#>"}
    inDescription : STRING(254);
    (*~
        <docu>
            <summary>
                Describes step status.
            </summary>
            <remarks>
                <para>
                    See <see cref="TcoCore.eStepStatus"/> for detailed description.
                </para>
            </remarks>
            enumStepStatus
        </docu>
    ~*)
    {attribute addProperty Name "<#Step status#>"}
    inStatus : eStepStatus;
    (*~
        <docu>
            <summary>
                Step duration time.
            </summary>
        </docu>
    ~*)
    {attribute addProperty Name "<#Step duration#>"}
    inDuration : TIME;
    (*~
        <docu>
            <summary>
                Total steps count;
            </summary>
        </docu>
    ~*)
    {attribute addProperty Name "<#Step count#>"}
    inStepCount : UINT;
END_VAR
END_METHOD

END_FUNCTION_BLOCK

// ---- POUs/Prototypes/TcoSequencer/TcoSequencer.TcPOU
FUNCTION_BLOCK PUBLIC ABSTRACT TcoSequencer EXTENDS TcoSequencerBase

(*~
    <docu>
        <summary>
            <para>
                Completes the sequencer, and return the sequencer pointer to the first step in the seuqence.
                Method is typically called inside the last step of the sequence.
            </para>
        </summary>
    </docu>
~*)
METHOD PROTECTED FINAL CompleteSequence
i_CompleteSequence();
END_METHOD

(*~
    <docu>
        <summary>
            Completes the execution of the current step and moves the sequencer pointer to the next step in order of execution.
            The call returns `ITcoObjectRestorer` that allows to restore object upon step completition.
        </summary>
        <returns></returns>
    </docu>
~*)
METHOD PROTECTED FINAL CompleteStep : ITcoObjectRestorer
CompleteStep := i_CompleteStep();
END_METHOD

(*~
    <docu>
        <summary>
            Terminates the currently executed step and set the sequencer's pointer to the step with Id that corresponds to ```inRequestedStepID``` parameter.
            When the order of the requested step is higher than the order of the currently finished step (the requested step is "after" the current one)
            the requested step is started in the same context cycle.
            When the order of the requested step is lower than the order of the currently finished step (the requested step is "before" the current one)
            the requested step is started in the next context cycle.
            If the requested step is not found even in the next context cycle, the sequencer enters error state ```StepWithRequestedIdDoesNotExists```.
            <para>
                See <see cref="TcoCore.eSequencerError"/> for detailed description.
            </para>
        </summary>
    </docu>
~*)
METHOD PROTECTED FINAL RequestStep : ITcoSequencer
VAR_INPUT
    (*~
        <docu>
            <summary>
                StepId of the step to be executed.
            </summary>
        </docu>
    ~*)
    inRequestedStepID : INT := MinStepID - 1;
END_VAR
VAR
    _message : STRING(254);
END_VAR
RequestStep := i_RequestStep(inRequestedStepID := inRequestedStepID);
END_METHOD

(*~
    <docu>
        <summary>
            <para>
                Ensures calling the Open(), Main() and Close() methods in the desired order.
                This method is final, so it cannot be overloaded. The **Instance.Run()** needs to be called cyclically inside the appropriate context.
            </para>
        </summary>
    </docu>
~*)
METHOD PUBLIC FINAL Run
THIS^.i_Open();
THIS^.Main();
THIS^.i_Close();
END_METHOD

METHOD PROTECTED Step : BOOL
VAR_INPUT
    (*~
    <docu>
        <summary>
            StepId of the current step.
            <remarks>
                <note type="important">
                    This number must be unique throughout the complete sequence.
                    It must be a constant or numerical literal and it must not change during the life-time of the sequencer.
                </note>
            </remarks>
        </summary>
    </docu>
~*)
    inStepID : INT;
    (*~
    <docu>
        <summary>
            If this value is false, step body is not executed and execution is moved to the next enabled step.
        </summary>
    </docu>
~*)
    inEnabled : BOOL;
    (*~
    <docu>
        <summary>
            Step description text.
        </summary>
    </docu>
~*)
    inStepDescription : STRING(254);
END_VAR
Step := i_Step(inStepID := inStepID, inEnabled := inEnabled, inStepDescription := inStepDescription);
END_METHOD

(*~
    <docu>
        <summary>
            Completes the actually running step, when the `inCondition` parameter is `TRUE`.
            Method is typically called inside a step as the transition method.
        </summary>
    </docu>
~*)
METHOD PROTECTED FINAL StepCompleteWhen
VAR_INPUT
    (*~
    <docu>
        <summary>
            The condition under which the step is completed.
        </summary>
    </docu>
~*)
    inCondition : BOOL;
END_VAR
i_StepCompleteWhen(inCondition := inCondition);
END_METHOD

END_FUNCTION_BLOCK

// ---- POUs/Prototypes/TcoSequencer/TcoSequencerObserver/TcoSequencerObserver.TcPOU
FUNCTION_BLOCK TcoSequencerObserver EXTENDS TcoObject IMPLEMENTS ITcoSequencerObserver
VAR
    _steps : ARRAY[0..MAX_STEPS] OF StepDetails;
    _currentStepOrder : UINT;
    _stepsCount : UINT;
END_VAR
VAR CONSTANT
    MAX_STEPS : UINT := 150;
END_VAR

{attribute 'hide'}
METHOD Clear : BOOL
VAR
    i : INT;
    blank : StepDetails;
END_VAR
{warning disable C0196}
FOR i := 0 TO MAX_STEPS DO
    {warning enable C0196}
    _steps[i] := blank;
END_FOR
END_METHOD

(*~
    <docu>
        <summary>
            Provides the mechanism to observe steps in the sequence and to gather basic infomation about step status and perfomance.
        </summary>
    </docu>
~*)
METHOD Observe
VAR_INPUT
    (*~
    <docu>
        <summary>
            Indicates that a step is active.
        </summary>
    </docu>
    ~*)
    inIsStepActive : BOOL;
    (*~
    <docu>
        <summary>
            Currently running step order.
        </summary>
    </docu>
    ~*)
    inCurrentStepOrder : UINT;
    (*~
    <docu>
        <summary>
            Step identification number.
        </summary>
        <remarks>
             <note type="important">
                This number must be unique throughout the complete sequence. It is required to uniquely identify the step of the sequence.
            </note>
            <para>
                The <see cref="PlcDocu.TcoCore.TcoSequencer.RequestStep"/> method is using this number to jump to the required step.
            </para>
        </remarks>
    </docu>
    ~*)
    {attribute addProperty Name "<#Step ID#>"}
    inID : INT;
    (*~
        <docu>
            <summary>
                Order of the step in the sequence.
            </summary>
        </docu>
    ~*)
    {attribute addProperty Name "<#Step Order#>"}
    inOrder : UINT;
    (*~
        <docu>
            <summary>
                If this value is false, step body is not executed and execution is moved to the next enabled step in the sequence.
            </summary>
        </docu>
    ~*)
    {attribute addProperty Name "<#Enabled#>"}
    inEnabled : BOOL;
    (*~
        <docu>
            <summary>
                Step description text.
            </summary>
        </docu>
    ~*)
    {attribute addProperty Name "<#Step description#>"}
    inDescription : STRING(254);
    (*~
        <docu>
            <summary>
                Describes step status.
            </summary>
            <remarks>
                <para>
                    See <see cref="TcoCore.eStepStatus"/> for detailed description.
                </para>
            </remarks>
            enumStepStatus
        </docu>
    ~*)
    {attribute addProperty Name "<#Step status#>"}
    inStatus : eStepStatus;
    (*~
        <docu>
            <summary>
                Step duration time.
            </summary>
        </docu>
    ~*)
    {attribute addProperty Name "<#Step duration#>"}
    inDuration : TIME;
    (*~
        <docu>
            <summary>
                Total steps count;
            </summary>
        </docu>
    ~*)
    {attribute addProperty Name "<#Step count#>"}
    inStepCount : UINT;
END_VAR
_currentStepOrder := inCurrentStepOrder;
_stepsCount := inStepCount;

IF (inOrder <= MAX_STEPS) THEN
    _steps[inOrder].ID := inID;
    _steps[inOrder].Order := inOrder;
    _steps[inOrder].Enabled := inEnabled;
    _steps[inOrder].Description := inDescription;

    IF (inCurrentStepOrder = inOrder) AND inIsStepActive THEN
        _steps[inOrder].Status := inStatus;
        _steps[inOrder].Duration := inDuration;
    END_IF;
END_IF;
END_METHOD

END_FUNCTION_BLOCK

// ---- POUs/Prototypes/TcoState/TcoState.TcPOU
FUNCTION_BLOCK TcoState EXTENDS TcoStateBase

METHOD PUBLIC ChangeState : ITcoState
VAR_INPUT
    NewState : INT;
END_VAR
ChangeState := SUPER^.ChangeStateProtected(NewState);
END_METHOD

(*~
    <docu>
        <summary>
            This method is called on each change of the <c>State</c>. This method could be overloaded and custom code should be placed here.
        </summary>
    </docu>
~*)
METHOD PROTECTED OnStateChange
VAR_INPUT
    PreviousState : INT;
    NewState : INT;
END_VAR
SUPER^.OnStateChange(PreviousState, NewState);
END_METHOD

END_FUNCTION_BLOCK

// ---- POUs/Prototypes/TcoStruct/TcoParentedStructure.TcPOU
FUNCTION_BLOCK TcoParentedStructure EXTENDS TcoObject

{attribute 'hide'}
METHOD FB_init : BOOL
VAR_INPUT
    bInitRetains : BOOL; // if TRUE, the retain variables are initialized (warm start / cold start)
    bInCopyCode : BOOL; // if TRUE, the instance afterwards gets moved into the copy code (online change)
    ParentObject : ITcoObject;
    ParentStruct : REFERENCE TO TcoStruct;
END_VAR
_Identity := ADR(THIS^);
_ParentObject := ParentObject;
_ParentStruct REF= ParentStruct;
END_METHOD

END_FUNCTION_BLOCK

// ---- POUs/Prototypes/TcoTask/TaskResult/TcoTaskResult.TcPOU
// credits Jakob Sagatowski https://github.com/sagatowski & contributors https://github.com/tcunit/TcUnit
FUNCTION_BLOCK TcoTaskResult
VAR
    _anyResult : ANY;
    F_AnyToUnionValue : F_AnyToUnionValue;
END_VAR

PROPERTY PUBLIC AsBool : BOOL
GET
Tc2_System.MEMCPY(destaddr := ADR(AsBool),
                  srcAddr := _anyResult.pValue,
                  n := _anyResult.diSize);
AsBool :=
END_GET
END_PROPERTY

METHOD PRIVATE Gee
VAR
    AnyValue : POINTER TO BYTE;
    AnySize : UDINT;
END_VAR
AnyValue := _anyResult.pValue;
AnySize := DINT_TO_UDINT(_anyResult.diSize);

CASE _anyResult.TypeClass OF
    IBaseLibrary.TypeClass.TYPE_BOOL:
        Tc2_System.MEMCPY(destaddr := ADR(F_AnyToUnionValue._bool), srcAddr := AnyValue, n := AnySize);
    IBaseLibrary.TypeClass.TYPE_BIT:
        {warning disable C0355}
        Tc2_System.MEMCPY(destaddr := ADR(F_AnyToUnionValue._bit), srcAddr := AnyValue, n := AnySize);
        {warning enable C0355}
    IBaseLibrary.TypeClass.TYPE_BYTE:
        Tc2_System.MEMCPY(destaddr := ADR(F_AnyToUnionValue._byte), srcAddr := AnyValue, n := AnySize);
    IBaseLibrary.TypeClass.TYPE_WORD:
        Tc2_System.MEMCPY(destaddr := ADR(F_AnyToUnionValue._word), srcAddr := AnyValue, n := AnySize);
    IBaseLibrary.TypeClass.TYPE_DWORD:
        Tc2_System.MEMCPY(destaddr := ADR(F_AnyToUnionValue._dword), srcAddr := AnyValue, n := AnySize);
    IBaseLibrary.TypeClass.TYPE_LWORD:
        Tc2_System.MEMCPY(destaddr := ADR(F_AnyToUnionValue._lword), srcAddr := AnyValue, n := AnySize);
    IBaseLibrary.TypeClass.TYPE_SINT:
        Tc2_System.MEMCPY(destaddr := ADR(F_AnyToUnionValue._sint), srcAddr := AnyValue, n := AnySize);
    IBaseLibrary.TypeClass.TYPE_INT:
        Tc2_System.MEMCPY(destaddr := ADR(F_AnyToUnionValue._int), srcAddr := AnyValue, n := AnySize);
    IBaseLibrary.TypeClass.TYPE_DINT:
        Tc2_System.MEMCPY(destaddr := ADR(F_AnyToUnionValue._dint), srcAddr := AnyValue, n := AnySize);
    IBaseLibrary.TypeClass.TYPE_LINT:
        Tc2_System.MEMCPY(destaddr := ADR(F_AnyToUnionValue._lint), srcAddr := AnyValue, n := AnySize);
    IBaseLibrary.TypeClass.TYPE_USINT:
        Tc2_System.MEMCPY(destaddr := ADR(F_AnyToUnionValue._usint), srcAddr := AnyValue, n := AnySize);
    IBaseLibrary.TypeClass.TYPE_UINT:
        Tc2_System.MEMCPY(destaddr := ADR(F_AnyToUnionValue._uint), srcAddr := AnyValue, n := AnySize);
    IBaseLibrary.TypeClass.TYPE_UDINT:
        Tc2_System.MEMCPY(destaddr := ADR(F_AnyToUnionValue._udint), srcAddr := AnyValue, n := AnySize);
    IBaseLibrary.TypeClass.TYPE_ULINT:
        Tc2_System.MEMCPY(destaddr := ADR(F_AnyToUnionValue._ulint), srcAddr := AnyValue, n := AnySize);
    IBaseLibrary.TypeClass.TYPE_REAL:
        Tc2_System.MEMCPY(destaddr := ADR(F_AnyToUnionValue._real), srcAddr := AnyValue, n := AnySize);
    IBaseLibrary.TypeClass.TYPE_LREAL:
        Tc2_System.MEMCPY(destaddr := ADR(F_AnyToUnionValue._lreal), srcAddr := AnyValue, n := AnySize);
    IBaseLibrary.TypeClass.TYPE_STRING:
        Tc2_System.MEMCPY(destaddr := ADR(F_AnyToUnionValue._string), srcAddr := AnyValue, n := AnySize);
    IBaseLibrary.TypeClass.TYPE_WSTRING:
        Tc2_System.MEMCPY(destaddr := ADR(F_AnyToUnionValue._wstring), srcAddr := AnyValue, n := AnySize);
    IBaseLibrary.TypeClass.TYPE_TIME:
        Tc2_System.MEMCPY(destaddr := ADR(F_AnyToUnionValue._time), srcAddr := AnyValue, n := AnySize);
    IBaseLibrary.TypeClass.TYPE_DATE:
        Tc2_System.MEMCPY(destaddr := ADR(F_AnyToUnionValue._date), srcAddr := AnyValue, n := AnySize);
    IBaseLibrary.TypeClass.TYPE_DATEANDTIME:
        Tc2_System.MEMCPY(destaddr := ADR(F_AnyToUnionValue._dateandtime), srcAddr := AnyValue, n := AnySize);
    IBaseLibrary.TypeClass.TYPE_TIMEOFDAY:
        Tc2_System.MEMCPY(destaddr := ADR(F_AnyToUnionValue._timeofday), srcAddr := AnyValue, n := AnySize);
    IBaseLibrary.TypeClass.TYPE_POINTER:
    (* None *)
    IBaseLibrary.TypeClass.TYPE_REFERENCE:
    (* None *)
    IBaseLibrary.TypeClass.TYPE_SUBRANGE:
    (* None *)
    IBaseLibrary.TypeClass.TYPE_ENUM:
    (* None *)
    IBaseLibrary.TypeClass.TYPE_ARRAY:
    (* None *)
    IBaseLibrary.TypeClass.TYPE_PARAMS:
    (* None *)
    IBaseLibrary.TypeClass.TYPE_USERDEF:
    (* None *)
    IBaseLibrary.TypeClass.TYPE_NONE:
    (* None *)
    IBaseLibrary.TypeClass.TYPE_ANY:
    (* None *)
    IBaseLibrary.TypeClass.TYPE_ANYBIT:
    (* None *)
    IBaseLibrary.TypeClass.TYPE_ANYDATE:
    (* None *)
    IBaseLibrary.TypeClass.TYPE_ANYINT:
    (* None *)
    IBaseLibrary.TypeClass.TYPE_ANYNUM:
    (* None *)
    IBaseLibrary.TypeClass.TYPE_ANYREAL:
    (* None *)
    IBaseLibrary.TypeClass.TYPE_LAZY:
    (* None *)
    IBaseLibrary.TypeClass.TYPE_LTIME:
        Tc2_System.MEMCPY(destaddr := ADR(F_AnyToUnionValue._ltime), srcAddr := AnyValue, n := AnySize);
    IBaseLibrary.TypeClass.TYPE_BITCONST:
    (* None *)
    IBaseLibrary.TypeClass.TYPE_INTERFACE:
(* None *)
ELSE
    (* None *)
END_CASE
END_METHOD

END_FUNCTION_BLOCK

// ---- POUs/Prototypes/TcoTier/TcoTier.TcPOU
{attribute 'hide'}
FUNCTION_BLOCK TcoTier EXTENDS TcoObject
VAR
    {attribute 'hide'}
    _nextExpectedCycle : ULINT;
END_VAR

{attribute 'hide'}
METHOD FB_init : BOOL
VAR_INPUT
    bInitRetains : BOOL; // if TRUE, the retain variables are initialized (warm start / cold start)
    bInCopyCode : BOOL; // if TRUE, the instance afterwards gets moved into the copy code (online change)
    ParentObject : ITcoObject;
END_VAR
END_METHOD

METHOD IsNewTier : BOOL
IsNewTier := THIS^.Context.StartCycleCount <> _nextExpectedCycle;
_nextExpectedCycle := THIS^.Context.StartCycleCount + 1;
END_METHOD

END_FUNCTION_BLOCK

// ---- POUs/Prototypes/TcoToggleTask/TcoToggleTask.TcPOU
(*~
    <docu>
        <summary>
            Provides basic toggling between two states. The states are triggered by calling the <see cref="PlcDocu.TcoCore.TcoToggleTask.Toggle()"/> method.
            <para>
                To get the actual state of the toggle task,
                <see cref="PlcDocu.TcoCore.TcoToggleTask.IsOn"/>,
                <see cref="PlcDocu.TcoCore.coToggleTask.IsOff"/>
                and <see cref="PlcDocu.TcoCore.TcoToggleTask.State"/> properties are available.
            </para>
        </summary>
    </docu>
~*)
{attribute addProperty StateOnDesc "<#On#>"}
{attribute addProperty StateOffDesc "<#Off#>"}
FUNCTION_BLOCK TcoToggleTask EXTENDS TcoObject IMPLEMENTS ITcoToggleTask
VAR
    {attribute clr [ReadOnly()]}
    _state : BOOL;
    (*~
    <docu>
        <summary>
            Use to toggle the state of this instance.
        </summary>
    </docu>
~*)
    {attribute addProperty Name "<#Toggle request#>"}
    _toggleRequest : BOOL;
    (*~
    <docu>
        <summary>
            Use to determine if the manipulation is enabled for example from the HMI application.
            This value is read only, to modify it use the property <see cref="PlcDocu.TcoCore.TcoToggleTask.Enabled()"/>
        </summary>
    </docu>
~*)
    {attribute addProperty Name "<#Enabled#>"}
    {attribute clr [ReadOnly()]}
    _enabled : BOOL := TRUE;
    {attribute 'hide'}
    _StartCycleCount : ULINT;
    (*~
    <docu>
        <summary>
            Indicated whether the task is in serviceable state. The default state 'serviceable' that means that the task
            can be invoked from the higher-level application. The serviceable state is cancelled when the immediate parent is `ITcoServiceable`
            and at the same time the parent is not in servicebable state. `TcoComponent` is serviceable, in order for the component's task to be
            invokable from higher-level application component must call `Service` method to induce the component into serviceable state.
        </summary>
    </docu>
    ~*)
    {attribute addProperty Name "<#Serviceable#>"}
    {attribute clr [ReadOnly()]}
    {attribute clr [RenderIgnore()]}
    _isServiceable : BOOL;
END_VAR

(*~
    <docu>
        <summary>
            Gets the context of this object.
            This context is given by declaration, its value is assigned after download by calling the implicit method <c>FB_init()</c> and cannot be changed during runtime.
        </summary>
    </docu>
~*)
PROPERTY Context : ITcoContext
GET
Context := THIS^.Parent.Context;
END_GET
END_PROPERTY

(*~
    <docu>
        <summary>
            Gets whether the any manipulation with this instance is enabled.
        </summary>
    </docu>
~*)
{attribute 'monitoring' := 'variable'}
PROPERTY Enabled : BOOL
GET
Enabled := _enabled;
END_GET
SET
_enabled := Enabled;
END_SET
END_PROPERTY

{attribute 'hide'}
METHOD PUBLIC FB_init : BOOL
VAR_INPUT
    bInitRetains : BOOL; // if TRUE, the retain variables are initialized (warm start / cold start)
    bInCopyCode : BOOL; // if TRUE, the instance afterwards gets moved into the copy code (online change)
    ParentObject : ITcoObject;
    InitState : BOOL;
END_VAR
_ParentObject := ParentObject;
_state := InitState;
END_METHOD

(*~
    <docu>
        <summary>
            Gets identity of this <see cref ="PlcDocu.TcoCore.TcoToggleTask()"/>.
            This value is assigned after download by calling the implicit method <c>FB_init()</c> and cannot be changed during runtime.
            This variable is used in the higher level applications.
        </summary>
    </docu>
~*)
PROPERTY Identity : ULINT
GET
Identity := _Identity;
END_GET
END_PROPERTY

{attribute 'monitoring' := 'variable'}
PROPERTY IsOff : BOOL
GET
IsOff := NOT _state;
END_GET
END_PROPERTY

{attribute 'monitoring' := 'variable'}
PROPERTY IsOn : BOOL
GET
IsOn := _state;
END_GET
END_PROPERTY

(*~
    <docu>
        <summary>
            Use to set the state of the '''TcoToggleTask''' to the value '''FALSE'''.
        </summary>
    </docu>
~*)
METHOD Off : BOOL
Off := FALSE;

//Check if Run method is called cyclically
IF THIS^.Context.StartCycleCount > _StartCycleCount + 1 THEN
    THIS^.Messenger.Programming('Run() method is not called cyclically.');
    RETURN;
END_IF

IF _enabled THEN
    IF _state THEN
        THIS^._state := FALSE;
        OnFtrig();
        OnStateChange();
        Off := TRUE;
    END_IF;
ELSE
    THIS^.Messenger.Post('Toggletask cannot be set to FALSE as its Enabled property is FALSE.', eMessageCategory.Info);
END_IF
END_METHOD

(*~
    <docu>
        <summary>
            Use to set the state of the '''TcoToggleTask''' to the value '''TRUE'''.
        </summary>
    </docu>
~*)
METHOD On : BOOL
On := FALSE;

//Check if Run method is called cyclically
IF THIS^.Context.StartCycleCount > _StartCycleCount + 1 THEN
    THIS^.Messenger.Programming('Run() method is not called cyclically.');
    RETURN;
END_IF

IF _enabled THEN
    IF NOT _state THEN
        THIS^._state := TRUE;
        OnRtrig();
        OnStateChange();
        On := TRUE;
    END_IF;
ELSE
    THIS^.Messenger.Post('Toggletask cannot be set to TRUE as its Enabled property is FALSE.', eMessageCategory.Info);
END_IF
END_METHOD

(*~
    <docu>
        <summary>
            Executes when toggle task changes its state from '''TRUE''' to '''FALSE'''.
        </summary>
    </docu>
~*)
METHOD PROTECTED OnFtrig
END_METHOD

(*~
    <docu>
        <summary>
            Executes when toggle task changes its state from '''FALSE''' to '''TRUE'''.
        </summary>
    </docu>
~*)
METHOD PROTECTED OnRtrig
END_METHOD

(*~
    <docu>
        <summary>
            Executes when toggle task changes its state .
        </summary>
    </docu>
~*)
METHOD PROTECTED OnStateChange
END_METHOD

(*~
    <docu>
        <summary>
            This method needs to be called cyclically.
        </summary>
    </docu>
~*)
METHOD Run
VAR
    _serviceableParent : ITcoServiceable;
END_VAR
// Store the context start cycle. Used to detect if Run() method is called cyclically.
_StartCycleCount := THIS^.Context.StartCycleCount;

// Detects if parent is in serviceable state to enable manual invoke of the task from the HMI/SCADA system.
IF (THIS^.Parent <> 0) THEN
    _isServiceable := TRUE;

    IF (__QUERYINTERFACE(THIS^.Parent, _serviceableParent)) THEN
        IF (NOT _serviceableParent.IsService) THEN
            THIS^._toggleRequest := FALSE;
            _isServiceable := FALSE;
        END_IF
    END_IF
END_IF;

//Triggering toggle
IF (THIS^._toggleRequest) THEN
    THIS^.Toggle();
END_IF;

THIS^._toggleRequest := FALSE;

IF _state THEN
    TaskOn();
ELSE
    TaskOff();
END_IF
END_METHOD

(*~
    <docu>
        <summary>
            Gets actual value of this instance.
        </summary>
    </docu>
~*)
{attribute 'monitoring' := 'variable'}
PROPERTY State : BOOL
GET
State := _state;
END_GET
END_PROPERTY

(*~
    <docu>
        <summary>
            Executes when toggle task is in ```Off``` state .
        </summary>
    </docu>
~*)
METHOD PROTECTED TaskOff
END_METHOD

(*~
    <docu>
        <summary>
            Executes when toggle task is in  ```On``` state .
        </summary>
    </docu>
~*)
METHOD PROTECTED TaskOn
END_METHOD

(*~
    <docu>
        <summary>
            Use to toggle the state of the '''TcoToggletask'''.
        </summary>
    </docu>
~*)
METHOD Toggle : BOOL
Toggle := FALSE;

//Check if Run method is called cyclically
IF THIS^.Context.StartCycleCount > _StartCycleCount + 1 THEN
    THIS^.Messenger.Programming('Run() method is not called cyclically.');
    RETURN;
END_IF

IF _enabled THEN
    THIS^._state := NOT THIS^._state;

    IF _state THEN
        OnRtrig();
    ELSE
        OnFtrig();
    END_IF

    OnStateChange();
    Toggle := TRUE;
ELSE
    THIS^.Messenger.Post('Toggletask cannot be triggered  as its Enabled property is FALSE.', eMessageCategory.Info);
END_IF
END_METHOD

END_FUNCTION_BLOCK

// ---- POUs/TestFixtures/_internals_TcoContext.TcPOU
{attribute 'hide'}
{attribute clr [ExcludeFromApiDocumentation()]}
FUNCTION_BLOCK ABSTRACT _internals_TcoContext EXTENDS TcoContext
VAR
    _probeCurrentCycleCount : ULINT;
    _probeRunRequiredCycles : ULINT;
    _testId : ULINT;
    _testDoneCounter : ULINT;
    _plcCycleCounter : ULINT;
END_VAR

{attribute 'TcRpcEnable'}
METHOD PROTECTED FINAL _Close
THIS^.Close();
END_METHOD

METHOD _GetSynchParams : RtcSynchParams
_GetSynchParams := RtcPrg._RtcSynchParams;
END_METHOD

{attribute 'TcRpcEnable'}
METHOD PROTECTED FINAL _Open
THIS^.Open();
END_METHOD

{attribute 'TcRpcEnable'}
METHOD PROTECTED FINAL _rtcUpdate
THIS^._rtc.UpdateInternal();
END_METHOD

METHOD ClearPlcCycleCounter
_plcCycleCounter := 0;
END_METHOD

METHOD ClearTestDoneCounter
_testDoneCounter := 0;
END_METHOD

METHOD ProbeDoneWhen
VAR_INPUT
    inCondition : BOOL;
END_VAR
IF inCondition THEN
    _testDoneCounter := _testDoneCounter + 1;
    _probeRunRequiredCycles := 0;
    _probeCurrentCycleCount := 0;
    {warning disable C0195}
    _testId := -1;
    {warning enable C0195}
END_IF
END_METHOD

METHOD ProbeRun
IF (_probeCurrentCycleCount < _probeRunRequiredCycles) THEN
    _plcCycleCounter := _plcCycleCounter + 1;
    SUPER^.Run();
    _probeCurrentCycleCount := _probeCurrentCycleCount + 1;
END_IF;
END_METHOD

END_FUNCTION_BLOCK

// ---- POUs/TestFixtures/_internals_TcoSequencer.TcPOU
{attribute 'hide'}
{attribute clr [ExcludeFromApiDocumentation()]}
FUNCTION_BLOCK ABSTRACT _internals_TcoSequencer EXTENDS TcoSequencer

{attribute 'hide'}
METHOD PROTECTED FINAL _Close
THIS^.i_Close();
END_METHOD

{attribute 'hide'}
METHOD PROTECTED FINAL _Open
THIS^.i_Open();
END_METHOD

END_FUNCTION_BLOCK

// ---- POUs/TestFixtures/_internals_TcoSequence.TcPOU
{attribute 'hide'}
{attribute clr [ExcludeFromApiDocumentation()]}
FUNCTION_BLOCK ABSTRACT _internals_TcoSequence EXTENDS TcoSequence

{attribute 'hide'}
METHOD PROTECTED FINAL _Close
THIS^.i_Close();
END_METHOD

{attribute 'hide'}
METHOD PROTECTED FINAL _Open
THIS^.i_Open();
END_METHOD

END_FUNCTION_BLOCK
